FUNCTION_BLOCK SS3_v_ps (* Composite FB wrapping other FBs *)
  (* Standard: 61499-2 *)
  (* Version 1.0, 2025-05-16, DEVIASH *)
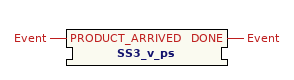
  EVENT_INPUT
    PRODUCT_ARRIVED;
  END_EVENT
  EVENT_OUTPUT
    DONE;
  END_EVENT
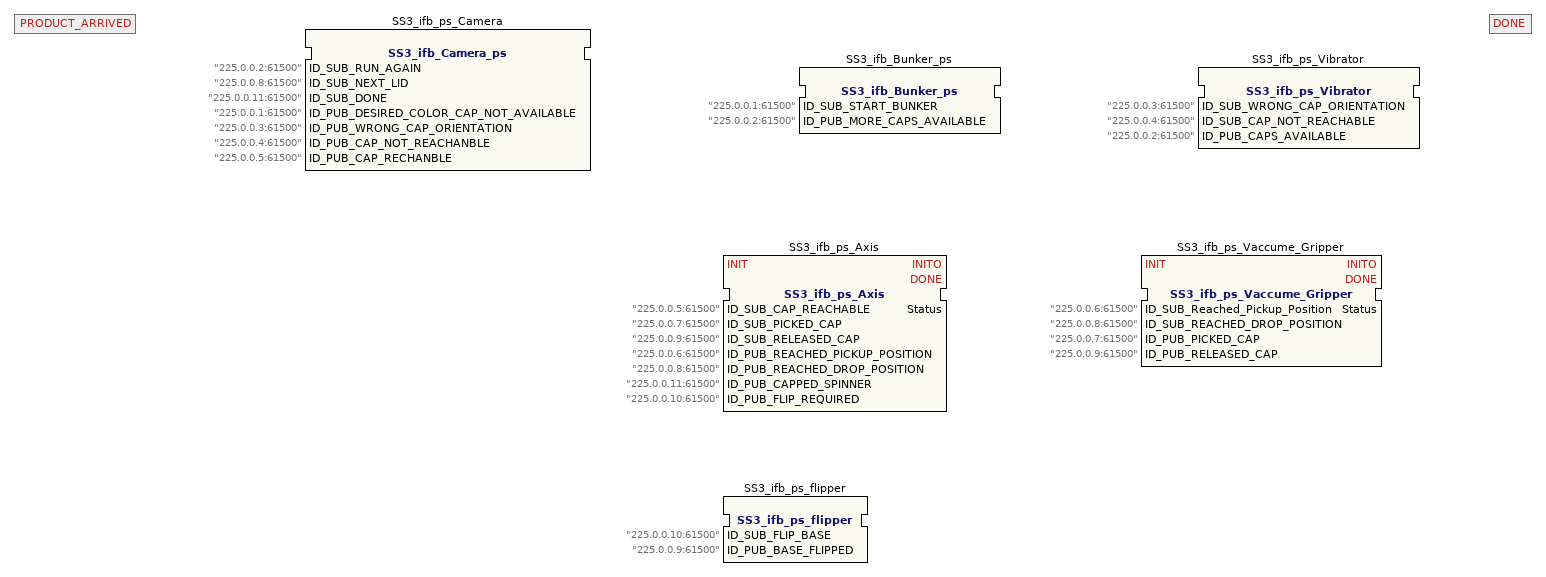
  FBS
    SS3_ifb_ps_Camera : SS3_ifb_Camera_ps(ID_SUB_RUN_AGAIN := "225.0.0.2:61500", ID_SUB_NEXT_LID := "225.0.0.8:61500", ID_SUB_DONE := "225.0.0.11:61500", ID_PUB_DESIRED_COLOR_CAP_NOT_AVAILABLE := "225.0.0.1:61500", ID_PUB_WRONG_CAP_ORIENTATION := "225.0.0.3:61500", ID_PUB_CAP_NOT_REACHANBLE := "225.0.0.4:61500", ID_PUB_CAP_RECHANBLE := "225.0.0.5:61500");
    SS3_ifb_ps_Vaccume_Gripper : SS3_ifb_ps_Vaccume_Gripper(ID_SUB_Reached_Pickup_Position := "225.0.0.6:61500", ID_SUB_REACHED_DROP_POSITION := "225.0.0.8:61500", ID_PUB_PICKED_CAP := "225.0.0.7:61500", ID_PUB_RELEASED_CAP := "225.0.0.9:61500");
    SS3_ifb_ps_Vibrator : SS3_ifb_ps_Vibrator(ID_SUB_WRONG_CAP_ORIENTATION := "225.0.0.3:61500", ID_SUB_CAP_NOT_REACHABLE := "225.0.0.4:61500", ID_PUB_CAPS_AVAILABLE := "225.0.0.2:61500");
    SS3_ifb_ps_flipper : SS3_ifb_ps_flipper(ID_SUB_FLIP_BASE := "225.0.0.10:61500", ID_PUB_BASE_FLIPPED := "225.0.0.9:61500");
    SS3_ifb_Bunker_ps : SS3_ifb_Bunker_ps(ID_SUB_START_BUNKER := "225.0.0.1:61500", ID_PUB_MORE_CAPS_AVAILABLE := "225.0.0.2:61500");
    SS3_ifb_ps_Axis : SS3_ifb_ps_Axis(ID_SUB_CAP_REACHABLE := "225.0.0.5:61500", ID_SUB_PICKED_CAP := "225.0.0.7:61500", ID_SUB_RELEASED_CAP := "225.0.0.9:61500", ID_PUB_REACHED_PICKUP_POSITION := "225.0.0.6:61500", ID_PUB_REACHED_DROP_POSITION := "225.0.0.8:61500", ID_PUB_CAPPED_SPINNER := "225.0.0.11:61500", ID_PUB_FLIP_REQUIRED := "225.0.0.10:61500");
  END_FBS
END_FUNCTION_BLOCK
